(* PLC project integracaoModBusTCPIP, Desconhecido Sem nome 1 *)
(* stored: creationDateTime 2023-12-06T19:26:37, modificationDateTime 2025-02-17T12:30:58 *)

PROGRAM planta
  VAR
    SP AT %QW0 : UINT := 50;  (* SetPoint *)
    PV AT %IW0 : UINT;  (* Sinal de entrada *)
    CV AT %QW1 : UINT := 0;  (* Sinal de controle *)
    ITERM AT %QD1 : REAL;
    error AT %QD2 : REAL;  (* Erro do sistema *)
    KP AT %QW2 : UINT := 3;  (* Contante Proporcional *)
    KI AT %QW3 : UINT := 13;  (* Ganho Integral *)
    R1 AT %IX0.0 : BOOL;  (* Reset bloco integração *)
  END_VAR
  VAR
    INTEGRAL0 : INTEGRAL;
  END_VAR

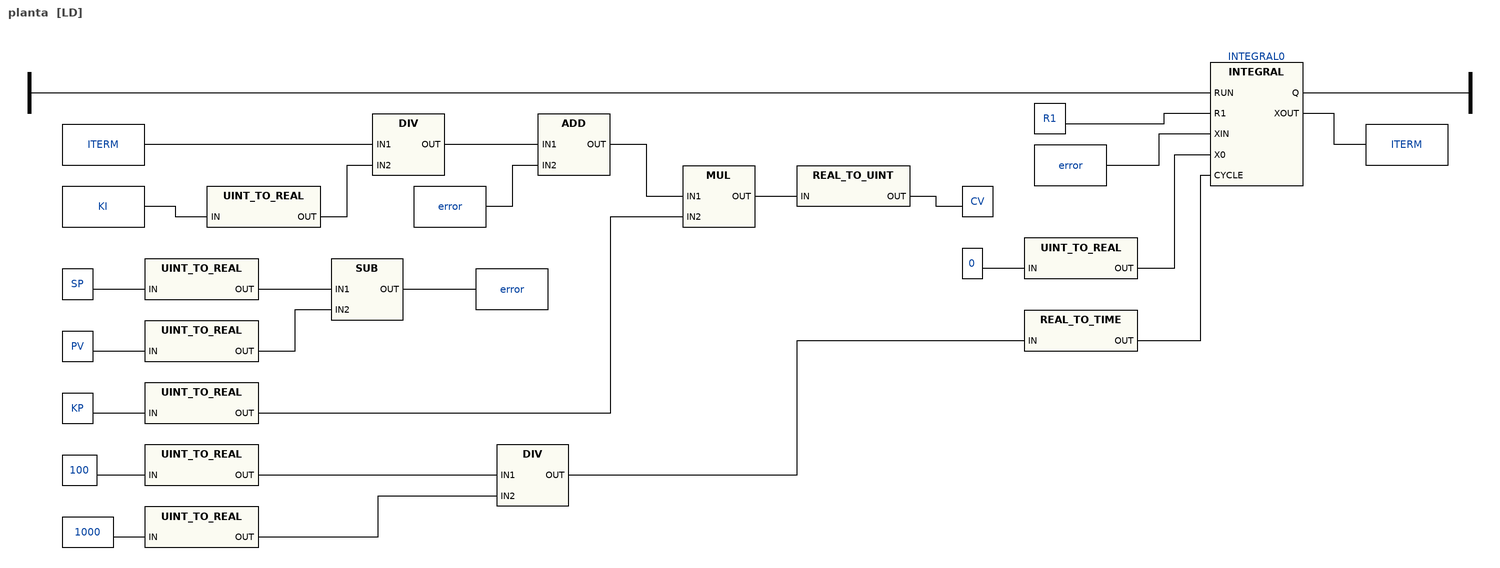
(* LD diagram, written out as Structured Text *)
CV := REAL_TO_UINT((ITERM / UINT_TO_REAL(KI) + error) * UINT_TO_REAL(KP));
error := UINT_TO_REAL(SP) - UINT_TO_REAL(PV);
INTEGRAL0(RUN := TRUE, R1 := R1, XIN := error, X0 := UINT_TO_REAL(0), CYCLE := REAL_TO_TIME(UINT_TO_REAL(100) / UINT_TO_REAL(1000)));
ITERM := INTEGRAL0.XOUT;
END_PROGRAM

CONFIGURATION Config0
  RESOURCE Res0 ON PLC
    TASK task0(INTERVAL := T#20ms, PRIORITY := 0);
    PROGRAM instance0 WITH task0 : planta;
  END_RESOURCE
END_CONFIGURATION
